// TIA Portal V20 export
FUNCTION "Program1" : Void   // FC1, LAD
{ S7_Optimized_Access := 'TRUE' }
// stored: SetENOAutomatically false
BEGIN

REGION Network 1
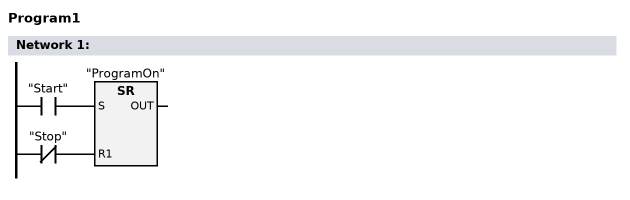
   RUNG wire#powerrail
      Contact( "Start" )
      S_SR(operand := "ProgramOn", r1 := wire#w1)
   END_RUNG
   RUNG wire#powerrail
      I_Contact( "Stop" )
   END_RUNG wire#w1
   // the same network as SCL:
   IF "Start" THEN
       "ProgramOn" := TRUE;   // SR flip-flop
   END_IF;
   IF NOT "Stop" THEN "ProgramOn" := FALSE; END_IF;
END_REGION
END_FUNCTION
